(* PLC project Test, D OpenPLC 1.0 *)
(* stored: creationDateTime 2018-09-26T00:48:44, modificationDateTime 2018-10-04T03:33:27 *)

PROGRAM Test_Program
  VAR
    ESP0 AT %QX0.0 : BOOL;
  END_VAR
  VAR
    TMP : BOOL;
  END_VAR
  VAR
    TMP0 AT %QX0.2 : BOOL;
    ESP1 AT %QX0.1 : BOOL;
  END_VAR

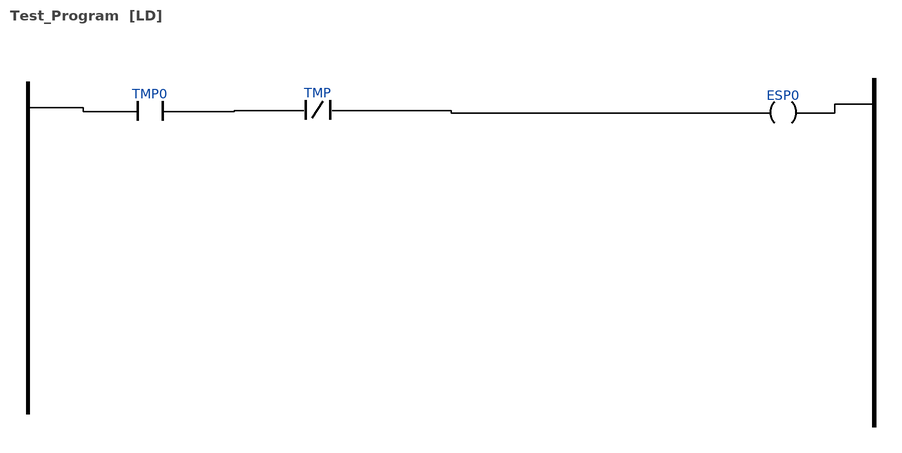
(* LD diagram, written out as Structured Text *)
ESP0 := TMP0 AND NOT TMP;
END_PROGRAM

CONFIGURATION Config0
  RESOURCE Res0 ON PLC
    TASK MyTask(INTERVAL := T#50ms, PRIORITY := 0);
    PROGRAM instance0 WITH MyTask : Test_Program;
  END_RESOURCE
END_CONFIGURATION
